Staubli VAL3: TrajBigBox.pjx

--- TrajBigBox.pjx ---
Parameters version=s7.6.3 stackSize=5000 millimeterUnit=true
Data file=TrajBigBox.dtx

--- TrajBigBox.dtx ---
public jointRx jToHome
public bool bMoveJHomeJoint = true
public num nIndexGun
public bool bJtEnabCheck[6] = true
public bool bPosEnabCheck[6]
  [0] = true
  [1] = true
  [2] = true
public num nRobCtrlAreaNum[12]
  [0] = -999
  [1] = 999
  [2] = -999
  [3] = 999
  [4] = -999
  [5] = 999
  [6] = -999
  [7] = 999
  [8] = -999
  [9] = 999
  [10] = -999
  [11] = 999
public num nRobCtrlHJtsNum[12]
  [0] = -180
  [1] = 180
  [2] = -130
  [3] = 147.5
  [4] = -145
  [5] = 145
  [6] = -270
  [7] = 270
  [8] = -115
  [9] = 140
  [10] = -270
  [11] = 270
